PROGRAM P01_AnalogScaling
VAR
	fbMixerSpeed				:FB_Scale;
	fbMixerSpeed2				:FB_Scale;
	fbMixerSpeed_AVG			:FB_AVG200;
	fbMixerCurrent				:FB_Scale;
	fbMixerCurrent_AVG			:FB_AVG200;
	
	fbChopper1Current			:FB_Scale;
	fbChopper1Current_AVG		:FB_AVG200;
	fbChopper2Current			:FB_Scale;
	fbChopper2Current_AVG		:FB_AVG200;
	
	fbProductTemperature		:FB_Scale;
	fbProductTemperature_AVG	:FB_AVG200;
	
	fbFlowMixerL				:FB_Scale;
	fbFlowMixerR				:FB_Scale;
	fbFlowChopper1				:FB_Scale;
	fbFlowChopper2				:FB_Scale;
	
	fbFlowMixerL_AVG			:FB_AVG200;
	fbFlowMixerR_AVG			:FB_AVG200;
	fbFlowChopper1_AVG			:FB_AVG200;
	fbFlowChopper2_AVG			:FB_AVG200;
	
	rOffset1					:REAL;
	fbChopper2Current2: FB_Scale;
	
	TON_SpeedRamp				:TON;
	tofMixerAV: TOF;
END_VAR

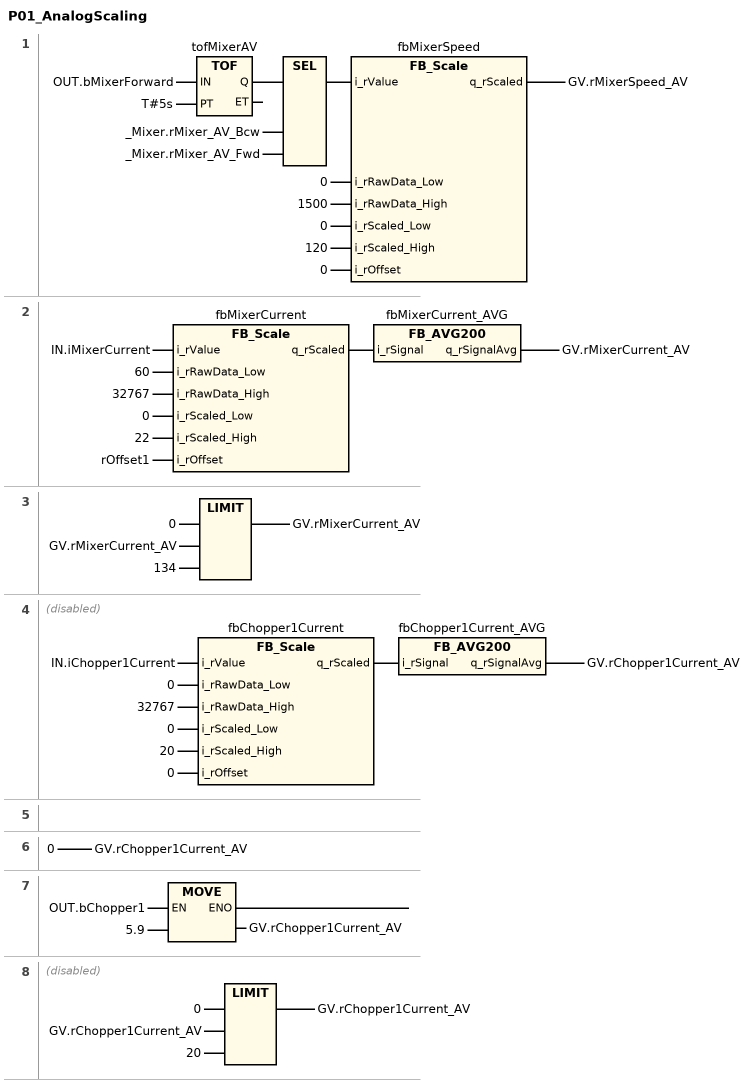
// NETWORK 1
tofMixerAV(IN := OUT.bMixerForward, PT := T#5s); // TOF
fbMixerSpeed(
    i_rValue := SEL(tofMixerAV.Q, _Mixer.rMixer_AV_Bcw, _Mixer.rMixer_AV_Fwd),
    i_rRawData_Low := 0,
    i_rRawData_High := 1500,
    i_rScaled_Low := 0,
    i_rScaled_High := 120,
    i_rOffset := 0); // FB_Scale
GV.rMixerSpeed_AV := fbMixerSpeed.q_rScaled;

// NETWORK 2
fbMixerCurrent(
    i_rValue := IN.iMixerCurrent,
    i_rRawData_Low := 60,
    i_rRawData_High := 32767,
    i_rScaled_Low := 0,
    i_rScaled_High := 22,
    i_rOffset := rOffset1); // FB_Scale
fbMixerCurrent_AVG(i_rSignal := fbMixerCurrent.q_rScaled); // FB_AVG200
GV.rMixerCurrent_AV := fbMixerCurrent_AVG.q_rSignalAvg;

// NETWORK 3
GV.rMixerCurrent_AV := LIMIT(0, GV.rMixerCurrent_AV, 134);

// NETWORK 4 (disabled)
// fbChopper1Current(
//     i_rValue := IN.iChopper1Current,
//     i_rRawData_Low := 0,
//     i_rRawData_High := 32767,
//     i_rScaled_Low := 0,
//     i_rScaled_High := 20,
//     i_rOffset := 0); // FB_Scale
// fbChopper1Current_AVG(i_rSignal := fbChopper1Current.q_rScaled); // FB_AVG200
// GV.rChopper1Current_AV := fbChopper1Current_AVG.q_rSignalAvg;

// NETWORK 5

// NETWORK 6
GV.rChopper1Current_AV := 0;

// NETWORK 7
IF OUT.bChopper1 THEN GV.rChopper1Current_AV := 5.9; END_IF

// NETWORK 8 (disabled)
// GV.rChopper1Current_AV := LIMIT(0, GV.rChopper1Current_AV, 20);

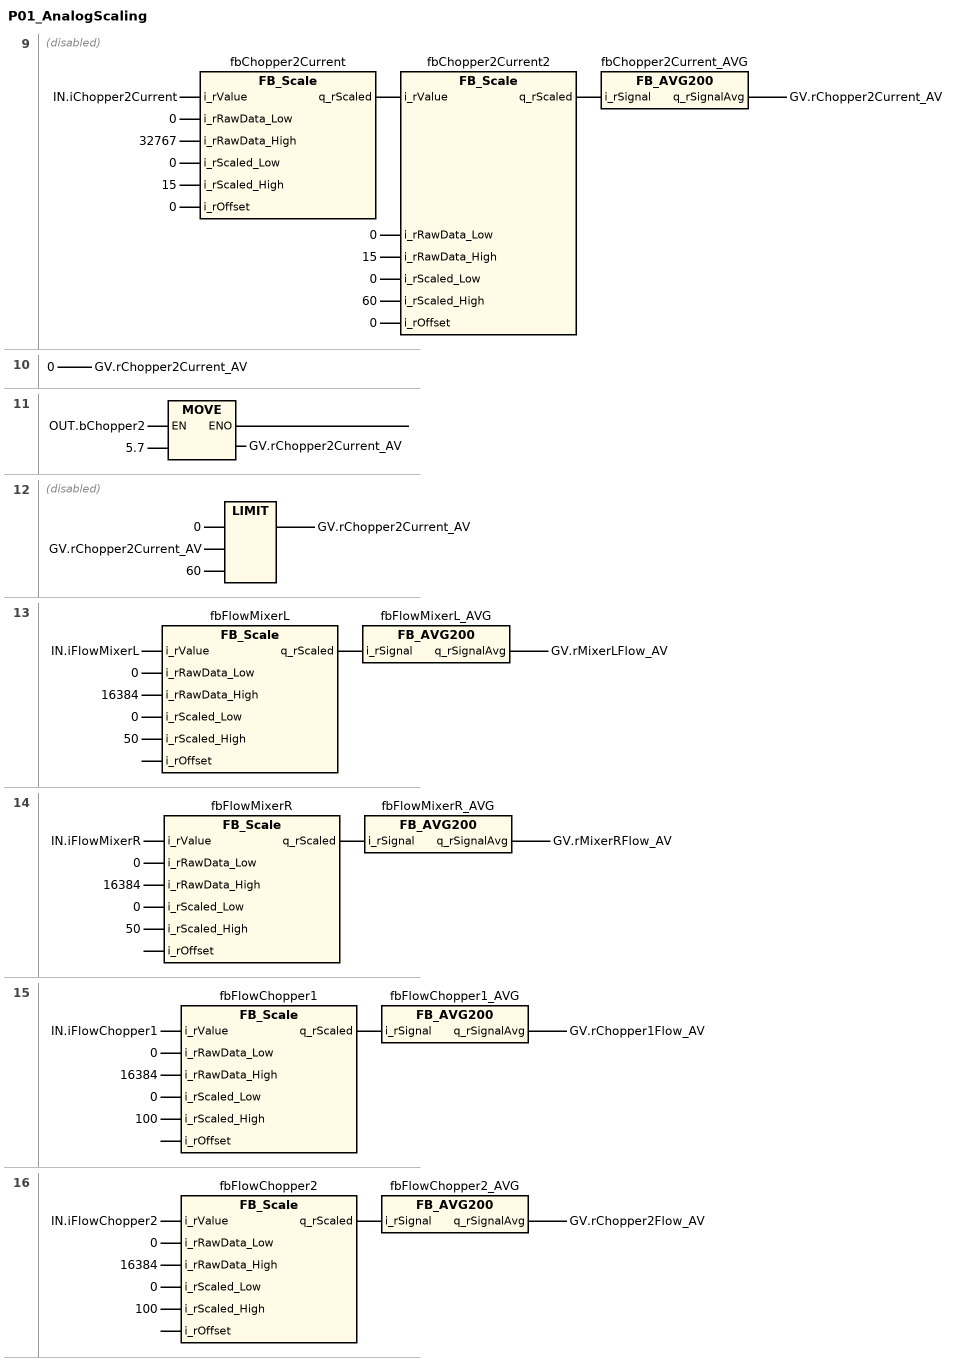
// NETWORK 9 (disabled)
// fbChopper2Current(
//     i_rValue := IN.iChopper2Current,
//     i_rRawData_Low := 0,
//     i_rRawData_High := 32767,
//     i_rScaled_Low := 0,
//     i_rScaled_High := 15,
//     i_rOffset := 0); // FB_Scale
// fbChopper2Current2(
//     i_rValue := fbChopper2Current.q_rScaled,
//     i_rRawData_Low := 0,
//     i_rRawData_High := 15,
//     i_rScaled_Low := 0,
//     i_rScaled_High := 60,
//     i_rOffset := 0); // FB_Scale
// fbChopper2Current_AVG(i_rSignal := fbChopper2Current2.q_rScaled); // FB_AVG200
// GV.rChopper2Current_AV := fbChopper2Current_AVG.q_rSignalAvg;

// NETWORK 10
GV.rChopper2Current_AV := 0;

// NETWORK 11
IF OUT.bChopper2 THEN GV.rChopper2Current_AV := 5.7; END_IF

// NETWORK 12 (disabled)
// GV.rChopper2Current_AV := LIMIT(0, GV.rChopper2Current_AV, 60);

// NETWORK 13
fbFlowMixerL(
    i_rValue := IN.iFlowMixerL,
    i_rRawData_Low := 0,
    i_rRawData_High := 16384,
    i_rScaled_Low := 0,
    i_rScaled_High := 50); // FB_Scale
fbFlowMixerL_AVG(i_rSignal := fbFlowMixerL.q_rScaled); // FB_AVG200
GV.rMixerLFlow_AV := fbFlowMixerL_AVG.q_rSignalAvg;

// NETWORK 14
fbFlowMixerR(
    i_rValue := IN.iFlowMixerR,
    i_rRawData_Low := 0,
    i_rRawData_High := 16384,
    i_rScaled_Low := 0,
    i_rScaled_High := 50); // FB_Scale
fbFlowMixerR_AVG(i_rSignal := fbFlowMixerR.q_rScaled); // FB_AVG200
GV.rMixerRFlow_AV := fbFlowMixerR_AVG.q_rSignalAvg;

// NETWORK 15
fbFlowChopper1(
    i_rValue := IN.iFlowChopper1,
    i_rRawData_Low := 0,
    i_rRawData_High := 16384,
    i_rScaled_Low := 0,
    i_rScaled_High := 100); // FB_Scale
fbFlowChopper1_AVG(i_rSignal := fbFlowChopper1.q_rScaled); // FB_AVG200
GV.rChopper1Flow_AV := fbFlowChopper1_AVG.q_rSignalAvg;

// NETWORK 16
fbFlowChopper2(
    i_rValue := IN.iFlowChopper2,
    i_rRawData_Low := 0,
    i_rRawData_High := 16384,
    i_rScaled_Low := 0,
    i_rScaled_High := 100); // FB_Scale
fbFlowChopper2_AVG(i_rSignal := fbFlowChopper2.q_rScaled); // FB_AVG200
GV.rChopper2Flow_AV := fbFlowChopper2_AVG.q_rSignalAvg;

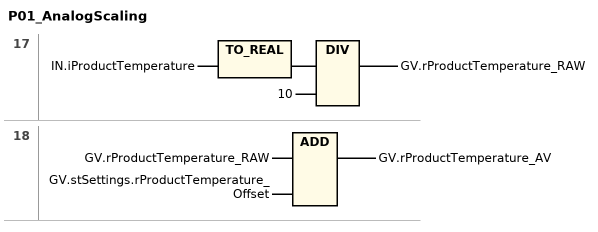
// NETWORK 17
GV.rProductTemperature_RAW := TO_REAL(IN.iProductTemperature) / 10;

// NETWORK 18
GV.rProductTemperature_AV := GV.rProductTemperature_RAW + GV.stSettings.rProductTemperature_Offset;

END_PROGRAM

(* stored: Version 1.1.0.1
   POU P01_AnalogScaling: Id {886e6b80-c86b-4d19-b9e4-45dd208fbc7d}, SpecialFunc None *)
